FUNCTION_BLOCK DigestTest
VAR_INPUT
END_VAR
VAR_OUTPUT
END_VAR
VAR
	un : STRING;
	pw : STRING;
	realm : STRING;
	meth : STRING;
	uri : STRING;
	qop : STRING;
	nonce : STRING;
	cnonce : STRING;
	nc : STRING;
	
	tempString : STRING(1000);
	
	retVal: BOOL;
	
	h1_byArr: ARRAY[0..15] OF BYTE;
	h1_hexStr: STRING;
	h2_byArr: ARRAY[0..15] OF BYTE;
	h2_hexStr: STRING;
	response_byArr: ARRAY[0..15] OF BYTE;
	response_hexStr: STRING;
	
	calculateNow : BOOL;
	i: INT;
END_VAR



IF calculateNow THEN
	
	// Values collected via wireshark
	un := 'Default User';
	pw := 'robotics';
	realm := 'validusers@robapi.abb';
	meth := 'GET';
	uri := '/rw/rapid/execution';
	qop := 'auth';
	nonce := 'MGY0Yjc2MGY2Y2QyZjAwNzp2YWxpZHVzZXJzQHJvYmFwaS5hYmI6MTkwMjg5NjRlNGE6MA==';
	cnonce := 'diddLOPR';
	nc := '00000001';
	
	
	tempString := '';
	tempString := CONCAT(tempString, un);
	tempString := CONCAT(tempString, ':');
	tempString := CONCAT(tempString, realm);
	tempString := CONCAT(tempString, ':');
	tempString := CONCAT(tempString, pw);
	
	retVal := F_GenerateHashValue(E_HashMode.HASH_MD5, ADR(tempString), LEN(tempString), ADR(h1_byArr), SIZEOF(h1_byArr));
	
	//h1_hexStr := DATA_TO_HEXSTR(ADR(h1_byArr), SIZEOF(h1_byArr), TRUE); // this method adds unnecessary space characters between bytes
	h1_hexStr := '';
	FOR i := 0 TO 15 DO
		h1_hexStr := CONCAT(h1_hexStr, BYTE_TO_HEXSTR(h1_byArr[i], 2, TRUE));
	END_FOR
	// expected value: 952890790eb23290847e6f4d57e76d86
	
	
	tempString := '';
	tempString := CONCAT(tempString, meth);
	tempString := CONCAT(tempString, ':');
	tempString := CONCAT(tempString, uri);
	
	retVal := F_GenerateHashValue(E_HashMode.HASH_MD5, ADR(tempString), LEN(tempString), ADR(h2_byArr), SIZEOF(h2_byArr));
	
	h2_hexStr := '';
	FOR i := 0 TO 15 DO
		h2_hexStr := CONCAT(h2_hexStr, BYTE_TO_HEXSTR(h2_byArr[i], 2, TRUE));
	END_FOR
	// expected value: 30bb6c0952d8c10cb9b2240a3772c67b
	
	
	tempString := '';
	tempString := CONCAT(tempString, h1_hexStr);
	tempString := CONCAT(tempString, ':');
	tempString := CONCAT(tempString, nonce);
	tempString := CONCAT(tempString, ':');
	tempString := CONCAT(tempString, nc);
	tempString := CONCAT(tempString, ':');
	tempString := CONCAT(tempString, cnonce);
	tempString := CONCAT(tempString, ':');
	tempString := CONCAT(tempString, qop);
	tempString := CONCAT(tempString, ':');
	tempString := CONCAT(tempString, h2_hexStr);
	
	retVal := F_GenerateHashValue(E_HashMode.HASH_MD5, ADR(tempString), LEN(tempString), ADR(response_byArr), SIZEOF(response_byArr));
	
	response_hexStr := '';
	FOR i := 0 TO 15 DO
		response_hexStr := CONCAT(response_hexStr, BYTE_TO_HEXSTR(response_byArr[i], 2, TRUE));
	END_FOR
	// expected value: c36e30cdd2961584cd41f6f49f6bcbba
	
	
	
	calculateNow := FALSE;
END_IF

END_FUNCTION_BLOCK

(* stored: Version 1.1.0.1, ProductVersion 3.1.4024.12
   POU DigestTest: Id {d5c05ab6-d9dc-4903-b1b4-a1d364a61d48}, SpecialFunc None *)
